// TIA Portal V19 export
DATA_BLOCK "Conveyor_RPM_to_MPM_DB"   // DB22
// stored: AutoNumber false, InstanceOfName RPM_to_MPM, InstanceOfType FB
"RPM_to_MPM"
   // VAR_INPUT
   //    RPM : LReal;
   //    Diameter : LReal;
   // END_VAR
   // VAR_OUTPUT
   //    MRM : Int;
   // END_VAR
BEGIN
END_DATA_BLOCK
